// TIA Portal project "JAVA GRUA" (V11)

(* hardware
DEVICE "S7300/ET200 station_1"  SIMATIC 300-Station
   slot 0: "Perfil soporte_0"  Rail  6ES7 390-1***0-0AA0
   slot 2: "PLC_1"  CPU 313C-2 DP  6ES7 313-6CF03-0AB0  V2.6
      slot 0: "Interfaz MPI_1"  MPI
      slot 1: "Interfaz DP_1"  DP
      slot 2: "DI16/DO16_1"  DI16/DO16
      slot 4: "Contaje_1"  Counter
*)

// ===== PLC "PLC_1"  CPU 313C-2 DP =====

VAR_GLOBAL   // PLC tag table "Tabla de variables estándar"
   "Tag_1" AT %A0.0 : Bool;
   "Tag_2" AT %A0.1 : Bool;
   "Tag_3" AT %A0.2 : Bool;
   "Tag_4" AT %A0.3 : Bool;
   "Tag_5" AT %A0.4 : Bool;
   "Tag_6" AT %E0.0 : Bool;
   "Tag_7" AT %E0.1 : Bool;
   "Tag_8" AT %E0.2 : Bool;
   "Tag_9" AT %E0.3 : Bool;
   "Tag_10" AT %E0.4 : Bool;
   "Tag_11" AT %E0.5 : Bool;
   "Tag_12" AT %E0.6 : Bool;
   "Tag_13" AT %E0.7 : Bool;
   "Tag_14" AT %E1.0 : Bool;
END_VAR

DATA_BLOCK "GRUA_DB"   // DB1
{ S7_Optimized_Access := 'FALSE' }
VERSION : 0.1
// stored: InstanceOfName GRUA
"GRUA"
BEGIN
END_DATA_BLOCK

FUNCTION_BLOCK "GRUA"   // FB1, SCL
{ S7_Optimized_Access := 'FALSE' }
VERSION : 0.1
   VAR_INPUT
      arriba : Bool;
      abajo : Bool;
      izquierda : Bool;
      derecha : Bool;
      paro : Bool;
      "FC ARRIBA" : Bool;
      "FC ABAJO" : Bool;
      "FC I" : Bool;
      "FC D" : Bool;
   END_VAR
   VAR_OUTPUT
      "m1 subir" : Bool;
      "m1 bajar" : Bool;
      "m2 izquierda" : Bool;
      "m2 derecha" : Bool;
   END_VAR
BEGIN
   IF #paro THEN
     #"m1 subir":=FALSE;
     #"m1 bajar":=FALSE;
     #"m2 derecha":=FALSE;
     #"m2 izquierda":=FALSE;
     RETURN;
   END_IF;

   IF #arriba AND NOT #"FC ARRIBA"AND NOT #"m1 bajar" THEN
     #"m1 subir":=true;
     #"m1 bajar":=false;
   ELSE
     #"m1 bajar":=false;
     #"m1 subir":= false   ;
     END_IF;

   IF #abajo AND NOT #"FC ABAJO" AND NOT #"m1 subir" THEN
      #"m1 bajar" :=true;
      #"m1 subir" :=false;
    END_IF;

   IF #arriba AND #abajo THEN
     #"m1 subir":=false;
     #"m1 bajar":=false;
   END_IF;

   IF #derecha AND NOT #"FC D" AND NOT #"m2 izquierda" THEN
     #"m2 derecha" :=true;
     #"m2 izquierda" :=false;
   ELSE
     #"m2 derecha" :=false;
     #"m2 izquierda" := false   ;
     END_IF;

   IF #izquierda AND NOT #"FC I" AND NOT #"m2 derecha" THEN
      #"m2 izquierda" :=true;
      #"m2 derecha" :=false;
    END_IF;

   IF #derecha AND #izquierda THEN
     #"m2 derecha" :=false;
     #"m2 izquierda" :=false;
     END_IF;
END_FUNCTION_BLOCK

ORGANIZATION_BLOCK "Main"   // OB1, LAD
TITLE = "Main Program Sweep (Cycle)"
{ S7_Optimized_Access := 'FALSE' }
VERSION : 0.1
   VAR_TEMP
      OB1_EV_CLASS : Byte;   // Bits 0-3 = 1 (Coming event), Bits 4-7 = 1 (Event class 1)
      OB1_SCAN_1 : Byte;   // 1 (Cold restart scan 1 of OB 1), 3 (Scan 2-n of OB 1)
      OB1_PRIORITY : Byte;   // Priority of OB Execution
      OB1_OB_NUMBR : Byte;   // 1 (Organization block 1, OB1)
      OB1_RESERVED_1 : Byte;   // Reserved for system
      OB1_RESERVED_2 : Byte;   // Reserved for system
      OB1_PREV_CYCLE : Int;   // Cycle time of previous OB1 scan (milliseconds)
      OB1_MIN_CYCLE : Int;   // Minimum cycle time of OB1 (milliseconds)
      OB1_MAX_CYCLE : Int;   // Maximum cycle time of OB1 (milliseconds)
      OB1_DATE_TIME : Date_And_Time;   // Date and time OB1 started
   END_VAR
BEGIN

REGION Network 1
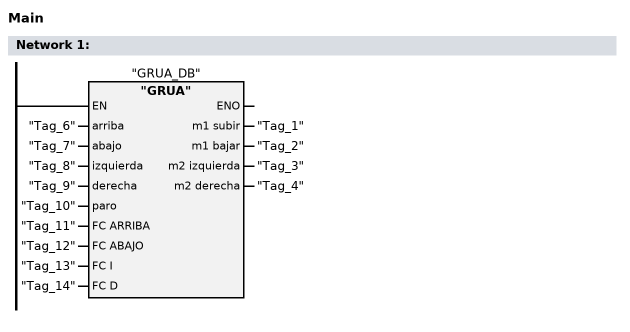
   RUNG wire#powerrail
      "GRUA_DB"(arriba := "Tag_6", abajo := "Tag_7", izquierda := "Tag_8", derecha := "Tag_9", paro := "Tag_10", "FC ARRIBA" := "Tag_11", "FC ABAJO" := "Tag_12", "FC I" := "Tag_13", "FC D" := "Tag_14", "m1 subir" => "Tag_1", "m1 bajar" => "Tag_2", "m2 izquierda" => "Tag_3", "m2 derecha" => "Tag_4")
   END_RUNG
   // the same network as SCL:
   "GRUA_DB"(arriba := "Tag_6",   // "GRUA"
             abajo := "Tag_7",
             izquierda := "Tag_8",
             derecha := "Tag_9",
             paro := "Tag_10",
             "FC ARRIBA" := "Tag_11",
             "FC ABAJO" := "Tag_12",
             "FC I" := "Tag_13",
             "FC D" := "Tag_14",
             "m1 subir" => "Tag_1",
             "m1 bajar" => "Tag_2",
             "m2 izquierda" => "Tag_3",
             "m2 derecha" => "Tag_4");
END_REGION
END_ORGANIZATION_BLOCK